{attribute 'GeneratedUsingTerminal: ELX9410-0000-0018'}
{attribute addProperty BoxType "ELX9410-0000-0018"}
{attribute addProperty Id "EtcSlaveTerminalBaseStatus_Us_InAT %I*Status_Us_In_B1E819A21Status_Us_OutAT %I*Status_Us_Out_B1E819A21WcStateAT %I*WcState_9091E0EB2InfoDataAT %I*InfoData_6F19DB2B2"}
{attribute addProperty CRC "3649559028"}
{attribute addProperty Size "6"}
TYPE ELX9410_D987D9F4 EXTENDS EtcSlaveTerminalBase :
STRUCT
	{attribute addProperty Name "Status_Us_In"}
	Status_Us_In : Status_Us_In_B1E819A2;
	{attribute addProperty Name "Status_Us_Out"}
	Status_Us_Out : Status_Us_Out_B1E819A2;
	{attribute addProperty Name "WcState"}
	WcState : WcState_9091E0EB;
	{attribute addProperty Name "InfoData"}
	InfoData : InfoData_6F19DB2B;
END_STRUCT
END_TYPE

(* stored: Version 1.2.0.0, ProductVersion 3.1.4024.9
   DUT ELX9410_D987D9F4: Id {f357223d-01f4-48eb-9158-a52ca5ce63ed} *)
